(* IEC 61131-3 sources: std_i2980_v2.06_cp053/Source/IMM/ieccontrol/SafetyGateGeneral, 1 file *)

(* ---- FBSafetyGateGeneral.pu ---- *)
IMPORT_OVER_LISTFILE
 tnSafetyGateState
, tevSafetyGateData
, tevSafetyGate
, tsDeviceId

END_IMPORT

FUNCTION_BLOCK FBSafetyGateGeneral #DUMMY_EDIT_BLOCK

VAR_INPUT
 bOpen : BOOL;
 bClosed : BOOL;
 dSupervisionTime : TIME;
END_VAR

VAR_OUTPUT
 State : tnSafetyGateState;
END_VAR

SYSTEM_VAR
 sv_DeviceId : tsDeviceId;
END_VAR

SYSTEM_OBJECT
 evSafetyGate : tevSafetyGate;
END_OBJECT

VAR
 evSafetyGateData : tevSafetyGateData;
END_VAR

(* IecGraph-Code *)

(* init step *)
INITIAL_STEP Step1:
END_STEP

(* steps *)
STEP CLOSED:
Action2 (P);
StateMessage (P);
END_STEP

ACTION Action2: #BEGIN_EDIT_BLOCK
State := nClosed

;#END_EDIT_BLOCK END_ACTION (*Action2*)
STEP OPEN:
Action4 (P);
StateMessage (P);
END_STEP

ACTION Action4: #BEGIN_EDIT_BLOCK
State := nOpen

;#END_EDIT_BLOCK END_ACTION (*Action4*)
STEP SUPERV:
Action5 (P);
StateMessage (P);
END_STEP

ACTION Action5: #BEGIN_EDIT_BLOCK
State := nOpen

;#END_EDIT_BLOCK END_ACTION (*Action5*)
STEP ERROR:
Action9 (P);
StateMessage (P);
END_STEP

ACTION Action9: #BEGIN_EDIT_BLOCK
State := nError

;#END_EDIT_BLOCK END_ACTION (*Action9*)
STEP STATE_CHANGED:
END_STEP

(* transitions *)
GO_ON_TRANSITION Trans1 FROM Step1 TO CLOSED :=  #BEGIN_EDIT_BLOCK
bClosed AND
NOT bOpen
;#END_EDIT_BLOCK
END_TRANSITION

TRANSITION Trans2 FROM CLOSED TO STATE_CHANGED :=  #BEGIN_EDIT_BLOCK
NOT bClosed OR
bOpen
;#END_EDIT_BLOCK
END_TRANSITION

GO_ON_TRANSITION Trans3 FROM Step1 TO OPEN :=  #BEGIN_EDIT_BLOCK
NOT bClosed AND
bOpen
;#END_EDIT_BLOCK
END_TRANSITION

TRANSITION Trans6 FROM OPEN TO STATE_CHANGED :=  #BEGIN_EDIT_BLOCK
bClosed OR
NOT bOpen
;#END_EDIT_BLOCK
END_TRANSITION

GO_ON_TRANSITION Trans4 FROM Step1 TO SUPERV :=  #BEGIN_EDIT_BLOCK
NOT (bClosed XOR bOpen)
;#END_EDIT_BLOCK
END_TRANSITION

TRANSITION Trans8 FROM SUPERV TO STATE_CHANGED :=  #BEGIN_EDIT_BLOCK
bClosed XOR bOpen
;#END_EDIT_BLOCK
END_TRANSITION

GO_ON_TRANSITION Trans9 FROM SUPERV TO ERROR :=  #BEGIN_EDIT_BLOCK
SUPERV.T >= dSupervisionTime
;#END_EDIT_BLOCK
END_TRANSITION

TRANSITION Trans11 FROM ERROR TO STATE_CHANGED :=  #BEGIN_EDIT_BLOCK
bClosed XOR bOpen
;#END_EDIT_BLOCK
END_TRANSITION

GO_ON_TRANSITION Trans5 FROM STATE_CHANGED TO Step1 :=  #BEGIN_EDIT_BLOCK
TRUE
;#END_EDIT_BLOCK
END_TRANSITION

(* end IecGraph-Code *)
(* sfc-code *)

(* stand alone actions *)
ACTION StateMessage: #BEGIN_EDIT_BLOCK
evSafetyGateData.DeviceId := sv_DeviceId;
evSafetyGateData.State := State;
SET_EVENT(evSafetyGate, evSafetyGateData);

;#END_EDIT_BLOCK END_ACTION (*StateMessage*)
(* end sfc-code *)

END_FUNCTION_BLOCK

#END_OF_IEC_PART

@Puma @IecEditor 6 30 @Pou 25
@@@BEG_Comment@@@

@@@END_Comment@@@

@BEG_Contents

@BEG_Func
@RT(17)FuncTreeContainer
0
@END_Func

@BEG_Const
@RT(18)ConstTreeContainer
0
@END_Const

@BEG_Export

@BEG_Kind
@FUNCTION_BLOCK @RT(19)FBSafetyGateGeneral @SEQUENTIAL_FLOW_CHART
@RT(0) @RT(0) @RT(0)
@END_Kind

@BEG_Dcl
@RT(16)DclTreeContainer
7
@Var @RT(5)bOpen @RT(0) @T @F @DT @RT(4)BOOL @RT(0) @T @T @BASIC 0 @F
@F @F
@T
@BEG_Attrib
3 @RT(0) @RT(0) @RT(0)
@END_Attrib
1 1 @F @F @F @F

@Var @RT(7)bClosed @RT(0) @T @F @DT @RT(4)BOOL @RT(0) @T @T @BASIC 0 @F
@F @F
@T
@BEG_Attrib
3 @RT(0) @RT(0) @RT(0)
@END_Attrib
1 1 @F @F @F @F

@Var @RT(16)dSupervisionTime @RT(0) @T @F @DT @RT(4)TIME @RT(0) @T @T @BASIC 0 @F
@F @F
@T
@BEG_Attrib
3 @RT(0) @RT(0) @RT(0)
@END_Attrib
1 1 @F @F @F @F

@Var @RT(5)State @RT(0) @T @T @DERIVED 0 @T @T @DT @RT(17)tnSafetyGateState @RT(0) @T @T @UNKNOWN 0 @F
@F @F
@T
@BEG_Attrib
3 @RT(0) @RT(0) @RT(0)
@END_Attrib
1 3 @F @F @F @F

@Var @RT(16)evSafetyGateData @RT(0) @T @T @DERIVED 0 @T @T @DT @RT(17)tevSafetyGateData @RT(0) @T @T @UNKNOWN 0 @F
@F @F
@T
@BEG_Attrib
3 @RT(0) @RT(0) @RT(0)
@END_Attrib
1 0 @F @F @F @F

@Var @RT(12)evSafetyGate @RT(0) @T @T @DERIVED 0 @T @T @DT @RT(13)tevSafetyGate @RT(0) @T @T @UNKNOWN 0 @F
@F @F
@T
@BEG_Attrib
3 @RT(0) @RT(0) @RT(0)
@END_Attrib
1 7 @F @F @F @F

@Var @RT(11)sv_DeviceId @RT(0) @T @T @DERIVED 0 @T @T @DT @RT(10)tsDeviceId @RT(0) @T @T @UNKNOWN 0 @F
@F @F
@T
@BEG_Attrib
3 @RT(0) @RT(0) @RT(0)
@END_Attrib
1 8 @F @F @F @F

@END_Dcl

@END_Export

@BEG_SfcBody
12 10 12

@BEG_SfcData 2
@StepSeq @RT(4)sseq @F 1
@Loop @RT(4)loop @F 2
@StepSeq @RT(3)seq @F 3
@Step @RT(5)Step1 @F @T @F @F @RT(0) @F
@AcbCont @RT(7)unnamed @F 0

@AltBranch @RT(3)alt @F 3
@TransSeq @RT(4)tseq @F 3
@Trans @RT(6)Trans1 @F @T @F @F @T @F @TL(3)
bClosed AND
NOT bOpen

@RT(6)Trans1 @F
@Step @RT(6)CLOSED @F @F @F @F @RT(0) @F
@AcbCont @RT(7)unnamed @F 2
@Acb @RT(7)Action2 @F @T @RT(1)P @RT(0) @F @F @T @TL(2)
State := nClosed

@F
@Acb @RT(12)StateMessage @F @F @RT(1)P @RT(0) @F @F @T @F

@Trans @RT(6)Trans2 @F @T @F @F @T @T @TL(3)
NOT bClosed OR
bOpen

@RT(6)Trans2 @F

@TransSeq @RT(4)tseq @F 3
@Trans @RT(6)Trans3 @F @T @F @F @T @F @TL(3)
NOT bClosed AND
bOpen

@RT(6)Trans3 @F
@Step @RT(4)OPEN @F @F @F @F @RT(0) @F
@AcbCont @RT(7)unnamed @F 2
@Acb @RT(7)Action4 @F @T @RT(1)P @RT(0) @F @F @T @TL(2)
State := nOpen

@F
@Acb @RT(12)StateMessage @F @F @RT(1)P @RT(0) @F @F @T @F

@Trans @RT(6)Trans6 @F @T @F @F @T @T @TL(3)
bClosed OR
NOT bOpen

@RT(6)Trans6 @F

@TransSeq @RT(4)tseq @F 3
@Trans @RT(6)Trans4 @F @T @F @F @T @F @TL(2)
NOT (bClosed XOR bOpen)

@RT(6)Trans4 @F
@Step @RT(6)SUPERV @F @F @F @F @RT(0) @F
@AcbCont @RT(7)unnamed @F 2
@Acb @RT(7)Action5 @F @T @RT(1)P @RT(0) @F @F @T @TL(2)
State := nOpen

@F
@Acb @RT(12)StateMessage @F @F @RT(1)P @RT(0) @F @F @T @F

@AltBranch @RT(3)alt @F 2
@TransSeq @RT(4)tseq @F 1
@Trans @RT(6)Trans8 @F @T @F @F @T @T @TL(2)
bClosed XOR bOpen

@RT(6)Trans8 @F

@TransSeq @RT(4)tseq @F 3
@Trans @RT(6)Trans9 @F @T @F @F @T @F @TL(2)
SUPERV.T >= dSupervisionTime

@RT(6)Trans9 @F
@Step @RT(5)ERROR @F @F @F @F @RT(0) @F
@AcbCont @RT(7)unnamed @F 2
@Acb @RT(7)Action9 @F @T @RT(1)P @RT(0) @F @F @T @TL(2)
State := nError

@F
@Acb @RT(12)StateMessage @F @F @RT(1)P @RT(0) @F @F @T @F

@Trans @RT(7)Trans11 @F @T @F @F @T @T @TL(2)
bClosed XOR bOpen

@RT(7)Trans11 @F

@Step @RT(13)STATE_CHANGED @F @F @F @F @RT(0) @F
@AcbCont @RT(7)unnamed @F 0

@Trans @RT(6)Trans5 @F @T @T @T @T @F @TL(2)
TRUE

@RT(6)Trans5 @F

@END_SfcData
@SaActions 1
@SaText @RT(12)StateMessage 1 @TL(4)
evSafetyGateData.DeviceId := sv_DeviceId;
evSafetyGateData.State := State;
SET_EVENT(evSafetyGate, evSafetyGateData);

@SaTrans 0
@SaExits 0
@END_SfcBody

@END_Contents
